FUNCTION TryConvert_UDINT_TO_ULINT : BOOL
VAR_INPUT
	in : UDINT;
	out : REFERENCE TO ULINT;
END_VAR

out := UDINT_TO_ULINT(in);
TryConvert_UDINT_TO_ULINT := TRUE;

END_FUNCTION

(* stored: Version 1.1.0.1, ProductVersion 3.1.4024.12
   POU TryConvert_UDINT_TO_ULINT: Id {4cb0aba8-8d85-4360-a3d4-408e9c1f6ddf}, SpecialFunc None *)
